{attribute 'GeneratedUsingTerminal: APS4322-7000-0017'}
{attribute addProperty BoxType "APS4322-7000-0017"}
{attribute addProperty Id "APS_InputsAT %I*APS_Inputs_4719D0DB98APS_DiagdataAT %I*APS_Diagdata_CE5B986F4APS_Comm_InputsAT %I*APS_Comm_Inputs_388FE28E10APS_OutputsAT %Q*APS_Outputs_31F2CBB3146APS_Comm_OutputsAT %Q*APS_Comm_Outputs_082002A44WcStateAT %I*WcState_9091E0EB2InfoDataAT %I*InfoData_BEF6B88E18"}
{attribute addProperty CRC "2093500820"}
{attribute addProperty Size "282"}
TYPE APS4322_7CC84994 EXTENDS EtcSlaveTerminalBase_947E5A46 :
STRUCT
	{attribute addProperty Name "APS_Inputs"}
	APS_Inputs : APS_Inputs_4719D0DB;
	{attribute addProperty Name "APS_Diagdata"}
	APS_Diagdata : APS_Diagdata_CE5B986F;
	{attribute addProperty Name "APS_Comm_Inputs"}
	APS_Comm_Inputs : APS_Comm_Inputs_388FE28E;
	{attribute addProperty Name "APS_Outputs"}
	APS_Outputs : APS_Outputs_31F2CBB3;
	{attribute addProperty Name "APS_Comm_Outputs"}
	APS_Comm_Outputs : APS_Comm_Outputs_082002A4;
	{attribute addProperty Name "WcState"}
	WcState : WcState_9091E0EB;
	{attribute addProperty Name "InfoData"}
	InfoData : InfoData_BEF6B88E;
END_STRUCT
END_TYPE

(* stored: Version 1.2.0.0, ProductVersion 3.1.4024.9
   DUT APS4322_7CC84994: Id {4272895b-66c4-4411-b798-52fd058b935c} *)
